# EPICS substitutions: ek9000App/Db/EL3101.substitutions
file EL3101.template
{       pattern
        {
                TERMINAL,

        }
        {
        }
}
